Fanuc TP program (LS listing): DOOR_COND.LS

/PROG  DOOR_COND	  Cond
/ATTR
OWNER		= MNEDITOR;
COMMENT		= "";
PROG_SIZE	= 210;
CREATE		= DATE 25-05-27  TIME 12:37:14;
MODIFIED	= DATE 25-05-27  TIME 12:45:14;
FILE_NAME	= T1_GRIP_;
VERSION		= 0;
LINE_COUNT	= 1;
MEMORY_SIZE	= 586;
PROTECT		= READ_WRITE;
TCD:  STACK_SIZE	= 0,
      TASK_PRIORITY	= 50,
      TIME_SLICE	= 0,
      BUSY_LAMP_OFF	= 0,
      ABORT_REQUEST	= 0,
      PAUSE_REQUEST	= 0;
DEFAULT_GROUP	= *,*,*,*,*;
CONTROL_CODE	= 00000000 00000000;
/APPL
/MN
   1:  WHEN DI[1110:OFF]=OFF,CALL DOOR_ERR ;
/POS
/END
